FUNCTION_BLOCK servo_validation

VAR_INPUT
offline_bit: BOOL;
error_bit: BOOL	;
servo_absolute: BOOL;
target_position: REAL;
servo_pos_delay_time: TIME;
END_VAR

VAR_OUTPUT
	servo_pos_delay_time_display: TIME;
	actual_position: REAL;
	absolute_done: BOOL;
END_VAR

VAR
	delay : ton;
END_VAR

// delay time move to timer
servo_pos_delay_time:=delay.PT;

// servo target position move to actual position
IF offline_bit AND NOT error_bit AND servo_absolute THEN
	delay.IN:=TRUE;
	IF delay.Q THEN
		absolute_done:=TRUE;
		actual_position:=target_position;
	END_IF
END_IF



// absolute done bit & timer in off
F_TRIG(CLK:=servo_absolute , Q=> );

IF f_trig.Q THEN
	absolute_done:=FALSE;
	delay.IN:=FALSE;
END_IF

END_FUNCTION_BLOCK

(* stored: Version 1.1.0.1, ProductVersion 3.1.4024.11
   POU servo_validation: Id {71bdb3eb-d897-4188-a63b-588ee923b08c}, SpecialFunc None *)
